Omron CX-Programmer project NewProject (CX-Programmer 9.73)

# PLC Simpang3: CP1H XA

## Global symbols (name address type ; comment)
0.00 BOOL  ; Start
0.01 BOOL  ; Stop
1000.01 BOOL  ; Lampu Kuning S1
100.00 BOOL  ; Lampu Hijau S1
100.01 BOOL  ; Lampu Kuning S1
100.02 BOOL  ; Lampu Merah S1
100.03 BOOL  ; Lampu Hijau S3
100.04 BOOL  ; Lampu Kuning S3
100.05 BOOL  ; Lampu Merah S3
100.06 BOOL  ; Lampu Hijau Lintas 2
100.07 BOOL  ; Lampu Merah Lintas 2
101.00 BOOL  ; Lampu Hijau Lintas 4
101.01 BOOL  ; Lampu Merah Lintas 4
101.02 BOOL  ; Lampu Merah Lintasan 5
101.03 BOOL  ; Lampu Hijau Lintasan 5
W0.00 BOOL  ; Running

## Program NewProgram1 (cyclic task 0)

### Section Section1

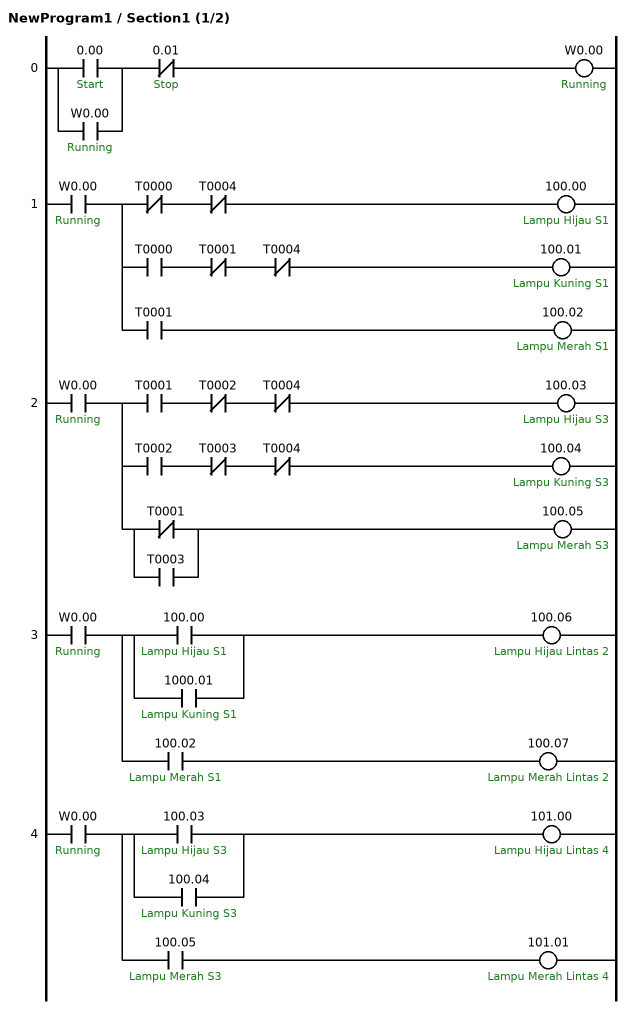
; rung 0
LD 0.00  ; Start
OR W0.00  ; Running
ANDNOT 0.01  ; Stop
OUT W0.00  ; Running
; rung 1
LD W0.00  ; Running
OUT TR0
ANDNOT T0000
ANDNOT T0004
OUT 100.00  ; Lampu Hijau S1
LD TR0
AND T0000
ANDNOT T0001
ANDNOT T0004
OUT 100.01  ; Lampu Kuning S1
LD TR0
AND T0001
OUT 100.02  ; Lampu Merah S1
; rung 2
LD W0.00  ; Running
OUT TR0
AND T0001
ANDNOT T0002
ANDNOT T0004
OUT 100.03  ; Lampu Hijau S3
LD TR0
AND T0002
ANDNOT T0003
ANDNOT T0004
OUT 100.04  ; Lampu Kuning S3
LD TR0
LDNOT T0001
OR T0003
ANDLD
OUT 100.05  ; Lampu Merah S3
; rung 3
LD W0.00  ; Running
OUT TR0
LD 100.00  ; Lampu Hijau S1
OR 1000.01  ; Lampu Kuning S1
ANDLD
OUT 100.06  ; Lampu Hijau Lintas 2
LD TR0
AND 100.02  ; Lampu Merah S1
OUT 100.07  ; Lampu Merah Lintas 2
; rung 4
LD W0.00  ; Running
OUT TR0
LD 100.03  ; Lampu Hijau S3
OR 100.04  ; Lampu Kuning S3
ANDLD
OUT 101.00  ; Lampu Hijau Lintas 4
LD TR0
AND 100.05  ; Lampu Merah S3
OUT 101.01  ; Lampu Merah Lintas 4

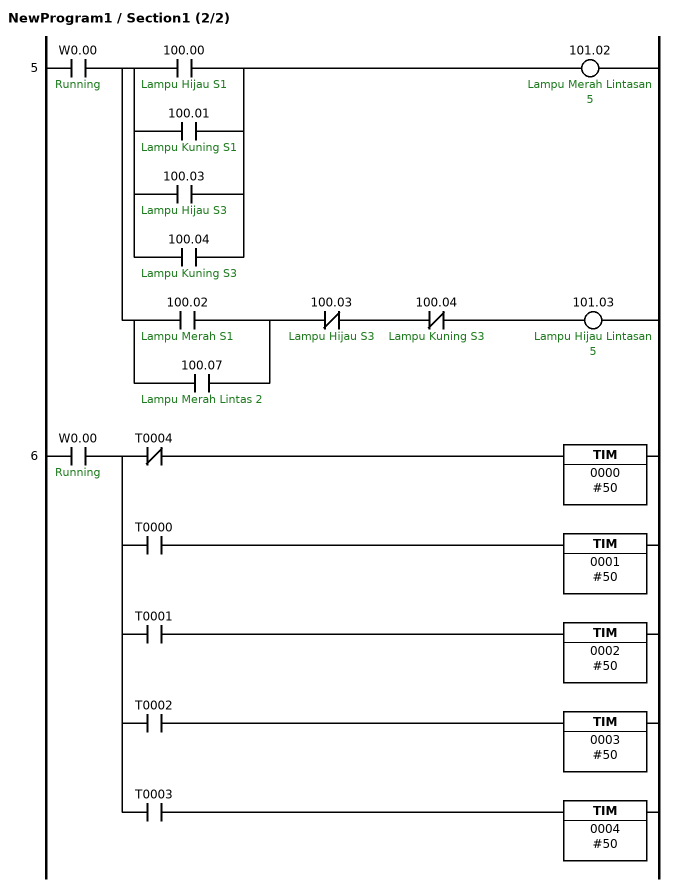
; rung 5
LD W0.00  ; Running
OUT TR0
LD 100.00  ; Lampu Hijau S1
OR 100.01  ; Lampu Kuning S1
OR 100.03  ; Lampu Hijau S3
OR 100.04  ; Lampu Kuning S3
ANDLD
OUT 101.02  ; Lampu Merah Lintasan 5
LD TR0
LD 100.02  ; Lampu Merah S1
OR 100.07  ; Lampu Merah Lintas 2
ANDLD
ANDNOT 100.03  ; Lampu Hijau S3
ANDNOT 100.04  ; Lampu Kuning S3
OUT 101.03  ; Lampu Hijau Lintasan 5
; rung 6
LD W0.00  ; Running
OUT TR0
ANDNOT T0004
TIM 0000 #50
LD TR0
AND T0000
TIM 0001 #50
LD TR0
AND T0001
TIM 0002 #50
LD TR0
AND T0002
TIM 0003 #50
LD TR0
AND T0003
TIM 0004 #50

### Section END
; rung 0
END(001)